TYPE ST_ExchangeData :
STRUCT
END_STRUCT
END_TYPE

(* stored: Version 1.1.0.1, ProductVersion 3.1.4026.8
   DUT ST_ExchangeData: Id {ed19bb78-b88c-498d-9a31-37fc83042cbb} *)
